Staubli VAL3: usrContinue.pgx

public program usrContinue(num& nWhichBttn (dimensions=1), bool bClear (dimensions=1))
begin
  if bClear
    cls()
    userPage()
    gotoxy(0,0)
    putln("                CONTINUE?")
    call usrButtonTxt(1,"NO")
    call usrButtonTxt(8,"YES")
  else
    putln("                CONTINUE?")
    call usrButtonTxt(1,"NO")
    call usrButtonTxt(8,"YES")
  endIf
  nWhichBttn=-1
  do
    nWhichBttn=(get()-270)
  until ((nWhichBttn==1) or (nWhichBttn==8))
end
